TYPE "TExtEncoder_Alarms"
VERSION : 0.1
// Block: TExtEncoder_Alarms
   STRUCT
      TOEncoder : Bool;
      MCFunction : Bool;
      TimeOutExecution : Bool;
   END_STRUCT;

END_TYPE
